// TIA Portal V17 export
// export: Created 2024-08-07T21:43:57.132572Z, ExportSetting WithDefaults, DisplayName Totally Integrated Automation Portal, DisplayVersion V17 Update 7, DisplayName TIA Portal Openness, DisplayVersion V17 Update 7, DisplayName TIA Portal Version Control Interface, DisplayVersion V17, DisplayName SINAMICS Startdrive Advanced, DisplayVersion V17 SP2, DisplayName SINAMICS Startdrive G110M, G120, G120C, G120D, G120P, G115D, DisplayVersion V17 SP2, DisplayName SINAMICS Startdrive G130, G150, S120, S150, SINAMICS MV, S210, DisplayVersion V17 SP2, DisplayName STEP 7 Professional, DisplayVersion V17 Update 7, DisplayName STEP 7 Safety, DisplayVersion V17 Update 6, DisplayName WinCC Advanced / Unified PC, DisplayVersion V17 Update 7
DATA_BLOCK "ServoMain_DB"   // DB6
VERSION : 0.1
// stored: AutoNumber true, DBAccessibleFromOPCUA true, DBAccessibleFromWebserver true, InstanceOfName ServoMain, InstanceOfType FB
"ServoMain"
   // VAR
   //    "TO_BasicPos_TA1-3MA_Instance" { S7_SetPoint := 'True'} : TO_BasicPos;
   //    IEC_Timer_0_Instance { S7_SetPoint := 'True'} : TON_TIME;
   //    "ServoControl_TA1-3MA_Instance" { S7_SetPoint := 'True'} : "ServoControl";
   //    IEC_Timer_0_Instance_1 { S7_SetPoint := 'True'} : TP_TIME;
   // END_VAR
BEGIN
END_DATA_BLOCK
